(* CODESYS project test2.project

Project tree, tasks and I/O mapping:
  Device : CODESYS Control Win V3, 3S - Smart Software Solutions GmbH, order no. 305021, version 3.5.8.10
    application Application
      libraries: Standard, * (System)
      task MainTask (cyclic, interval t#20ms, priority 1) calls PLC_PRG
      task VISU_TASK (cyclic, interval 100 ms, priority 31) calls VisuElems.Visu_Prg
      program PLC_PRG [ST]
      visualisation Visualization
  text list GlobalTextList
*)

// Device/Application/PLC_PRG
PROGRAM PLC_PRG
VAR
	t1: TON;
	zegar: BOOL;
	zmienna: TIME;
	
	przycisk1: BOOL;
	przycisk2: BOOL;
	przycisk3: BOOL;
	przycisk4: BOOL;
	przycisk5: BOOL;
	
	winda_na_1: BOOL;
	winda_na_5: BOOL;
	
	winda_1: BOOL;
	winda_5: BOOL;
	
	licznik: WORD;

	ctud1: CTUD;
	
	moveY: INT;
	
	nieaktywne: BOOL;

END_VAR

t1(IN:=zegar,PT:=T#0.1MS);
zmienna:=t1.ET;
zegar:=NOT(t1.Q);

ctud1(CU:=(zegar AND winda_5),CD:=(zegar AND winda_1),RESET:=FALSE,LOAD:=FALSE,PV:=360);
winda_na_5:=ctud1.QU;
winda_na_1:=ctud1.QD;
licznik:=ctud1.CV;


/////////////////////////////////////////////////////////////////////


IF (WORD_TO_INT(licznik) < moveY) THEN
	winda_5:=TRUE;
END_IF

IF (WORD_TO_INT(licznik) > moveY) THEN
	winda_1:=TRUE;
END_IF


/////////////////////////////////////////////////////////////////////


IF przycisk1=TRUE THEN
	moveY:=0;
END_IF

IF przycisk2=TRUE THEN
	moveY:=90;
END_IF

IF przycisk3=TRUE THEN
	moveY:=180;
END_IF

IF przycisk4=TRUE THEN
	moveY:=270;
END_IF

IF przycisk5=TRUE THEN
	moveY:=360;
END_IF


/////////////////////////////////////////////////////////////////////


IF (przycisk1=TRUE OR przycisk2=TRUE OR przycisk3=TRUE OR przycisk4=TRUE OR przycisk5=TRUE) THEN
	nieaktywne:=TRUE;
END_IF


/////////////////////////////////////////////////////////////////////


IF (licznik=0 AND przycisk1=TRUE) THEN
	przycisk1:=FALSE;
	nieaktywne:=FALSE;
	winda_1:=FALSE;
	winda_5:=FALSE;
END_IF

IF (licznik=90 AND przycisk2=TRUE) THEN
	przycisk2:=FALSE;
	nieaktywne:=FALSE;
	winda_1:=FALSE;
	winda_5:=FALSE;
END_IF

IF (licznik=180 AND przycisk3=TRUE) THEN
	przycisk3:=FALSE;
	nieaktywne:=FALSE;
	winda_1:=FALSE;
	winda_5:=FALSE;
END_IF

IF (licznik=270 AND przycisk4=TRUE) THEN
	przycisk4:=FALSE;
	nieaktywne:=FALSE;
	winda_1:=FALSE;
	winda_5:=FALSE;
END_IF

IF (licznik=360 AND przycisk5=TRUE) THEN
	przycisk5:=FALSE;
	nieaktywne:=FALSE;
	winda_1:=FALSE;
	winda_5:=FALSE;
END_IF

END_PROGRAM

// Device/Application/Visualization
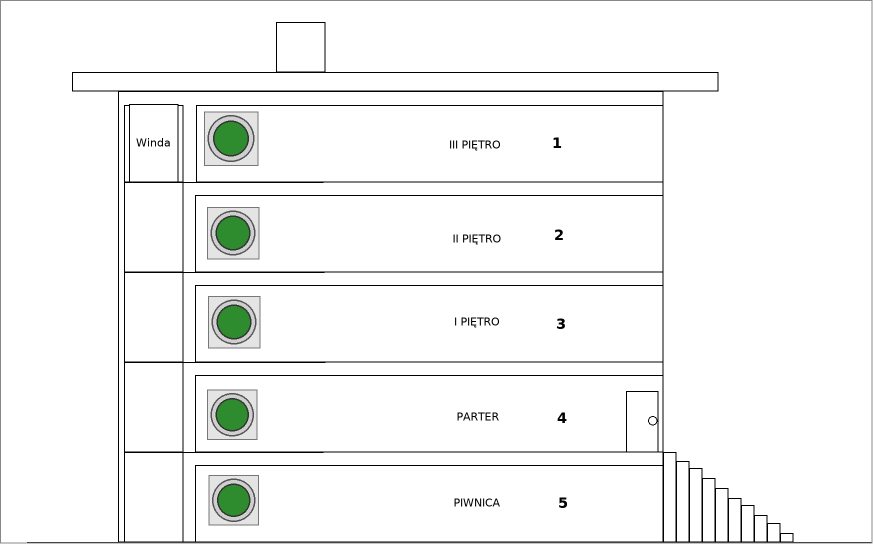
VISUALIZATION Visualization  // 873x544
    Rectangle (118,91 545x451)
    Rectangle (195,465 468x77)
    Rectangle (124,105 59x77)
    Rectangle (124,182 59x90)
    Rectangle (124,272 59x90)
    Rectangle (124,362 59x90)
    Rectangle (124,452 59x90)
    Rectangle (129,104 49x78), "Winda"
        p2738717112: PLC_PRG.licznik
    Rectangle (195,375 468x77)
    Rectangle (195,285 468x77)
    Rectangle (195,195 468x77)
    Rectangle (196,105 467x77)
    Rectangle (72,72 646x19)
    Rectangle (276,22 49x50)
    Line (672,542) (871,542)
    Rectangle (626,391 32x61)
    Rectangle (663,452 13x90)
    Rectangle (676,461 13x81)
    Rectangle (689,468 13x74)
    Rectangle (702,478 13x64)
    Rectangle (715,488 13x54)
    Rectangle (728,498 13x44)
    Rectangle (741,505 13x37)
    Rectangle (754,515 13x27)
    Rectangle (767,523 13x19)
    Rectangle (780,533 13x9)
    Line (27,542) (226,542)
    Line (124,452) (323,452)
    Line (126,362) (325,362)
    Line (125,272) (324,272)
    Line (124,182) (323,182)
    Ellipse (648,416 9x9)
    Label (402,488 150x30), "PIWNICA"
    Label (403,402 150x30), "PARTER"
    Label (402,307 150x30), "I PIĘTRO"
    Label (402,224 150x30), "II PIĘTRO"
    Label (400,130 150x30), "III PIĘTRO"
    PushSwitch (204,111 54x55), variable: PLC_PRG.przycisk1, input disabled if: PLC_PRG.nieaktywne, behaviour: TOGGLE, style: Switch-PushSwitch-Green
    PushSwitch (207,388 50x53), variable: PLC_PRG.przycisk4, input disabled if: PLC_PRG.nieaktywne, behaviour: TOGGLE, style: Switch-PushSwitch-Green
    PushSwitch (207,296 54x52), variable: PLC_PRG.przycisk3, input disabled if: PLC_PRG.nieaktywne, behaviour: TOGGLE, style: Switch-PushSwitch-Green
    PushSwitch (207,207 52x52), variable: PLC_PRG.przycisk2, input disabled if: PLC_PRG.nieaktywne, behaviour: TOGGLE, style: Switch-PushSwitch-Green
    PushSwitch (207,475 53x50), variable: PLC_PRG.przycisk5, input disabled if: PLC_PRG.nieaktywne, behaviour: TOGGLE, style: Switch-PushSwitch-Green
    Label (488,488 150x30), "5"
    Label (487,403 150x30), "4"
    Label (486,309 150x30), "3"
    Label (484,220 150x30), "2"
    Label (482,128 150x30), "1"
END_VISUALIZATION
